// TIA Portal V17 export
// export: Created 2024-09-02T12:50:34.1146728Z, ExportSetting WithDefaults, DisplayName Totally Integrated Automation Portal, DisplayVersion V17, DisplayName TIA Portal Openness, DisplayVersion V17, DisplayName TIA Portal Version Control Interface, DisplayVersion V17, DisplayName STEP 7 Professional, DisplayVersion V17, DisplayName STEP 7 Safety, DisplayVersion V17, DisplayName WinCC Professional, DisplayVersion V17
TYPE "TypeKeyData"
// stored: IsFailsafeCompliant false
   STRUCT
      EKSAdapterIndex : UInt;
      CostCenter : Array[0..3] of Char;
      DateEnd : Array[0..7] of Char;
      ProtectionLevel : Int;
      Operator_ID : Array[1..7] of Char;
      SafetyMode : Byte;
      Specialbits : Byte;
      SerialNumber : Array[1..8] of Byte;
      KeyAdapterReady : Bool;
      KeyDetected : Bool;
      ChecksumNotOK : Bool;
      DateNotOK : Bool;
      CostCenterNotOK : Bool;
      KeyDataNotOK : Bool;
      EKSKeyInvalidLess30Days : Bool;
   END_STRUCT;
END_TYPE
